PROGRAM PRG_TEST
VAR
    (*PrimitiveTypesTest : FB_PrimitiveTypes_Test;
    AssertTrueFalse_Test : FB_AssertTrueFalse_Test;
    AssertEveryFailedTestTwice : FB_AssertEveryFailedTestTwice;
    CreateFourTestsWithSameName : FB_CreateFourTestsWithSameName;
    ArrayPrimitiveTypes_Test : FB_ArrayPrimitiveTypes_Test;
    CreateDisabledTest : FB_CreateDisabledTest;
    AnyPrimitiveTypes_Test : FB_AnyPrimitiveTypes_Test;
    AssertEveryFailedTestTwice_ArrayVersion : FB_AssertEveryFailedTestTwice_ArrayVersion;
    AnyToUnionValue_Test : FB_AnyToUnionValue_Test;*)
    AnyToString_Test: FB_AnyToString_Test;
    SimpleStringBuilder_Test: FB_SimpleStringBuilder_Test;
    Printer_Test: FB_Printer_Test;
    Runner_Test: FB_Runner_Test;
    TestSuite_Test: FB_TestSuite_Test;
END_VAR

TcUnit.RUN();

END_PROGRAM

(* stored: Version 1.1.0.1, ProductVersion 3.1.4022.12
   POU PRG_TEST: Id {35d0cb91-f449-41c5-be41-3ca0dfe074f2}, SpecialFunc None *)
